{attribute 'qualified_only'}
VAR_GLOBAL
    ConveyorRunning : BOOL   := FALSE;
    MotorTemp       : REAL   := 72.5;
    PartCount       : INT    := 0;
END_VAR

(* stored: Version 1.1.0.1, ProductVersion 3.1.4026.18
   GVL MachineData: Id {97298d33-68ec-46b5-8207-508c529c95e8} *)
